# EPICS autosave request: iocBoot/iocUSB231/auto_settings.req
file "USB231_settings.req", P=USB231:
